{attribute 'reflection'} 
FUNCTION_BLOCK FB_Component EXTENDS FB_Cycle IMPLEMENTS I_Component
VAR_INPUT
	fbInfo:						FB_Info(sInstancePath);
	fbObserver:					FB_Observer;
	fbEvent:					FB_Event(THIS^);
END_VAR
VAR_OUTPUT
END_VAR
VAR
    {attribute 'hide'}
	{attribute 'instance-path'} 
    {attribute 'noinit'}
    sInstancePath:				STRING(255);	
	eRequest:					E_Request;
	eState:						E_State;
    {attribute 'hide'}
	eStatePrevious:				E_State;
END_VAR

METHOD PROTECTED M_Aborted : BOOL
VAR_INPUT
END_VAR
// State Aborted
M_Aborted:= True;
END_METHOD

METHOD PROTECTED M_Aborting : BOOL
VAR_INPUT
END_VAR
// State Aborting
M_Aborting:= True;
END_METHOD

METHOD PROTECTED M_Completed : BOOL
VAR_INPUT
END_VAR
// State Complete
M_Completed:= TRUE;
END_METHOD

METHOD PROTECTED M_Completing : BOOL
VAR_INPUT
END_VAR
// State Completing
M_Completing:= True;
END_METHOD

METHOD PUBLIC M_Cycle
VAR_INPUT
END_VAR
fbInfo();
fbObserver();
fbEvent();

// Handle Module Type Package states
CASE eState OF
	E_State.Undefined:
		IF M_Initialise() THEN
			eState:= E_State.Idle;					
		END_IF
		
	E_State.Resetting:
		CASE eRequest OF
			E_Request.Stop:
				eState:= E_State.Stopping;					
			E_Request.Abort:
				eState:= E_State.Aborting;						
		END_CASE	
		IF M_Resetting() THEN
			eState:= E_State.Idle;
		END_IF
		
	E_State.Idle:
		CASE eRequest OF
			E_Request.Start:
				eState:= E_State.Starting;
			E_Request.Stop:
				eState:= E_State.Stopping;					
			E_Request.Abort:
				eState:= E_State.Aborting;
			ELSE
				eRequest:= E_Request.Undefined;						
		END_CASE
		M_Idle();
		
	E_State.Starting:
		CASE eRequest OF
			E_Request.Stop:
				eState:= E_State.Stopping;					
			E_Request.Abort:
				eState:= E_State.Aborting;				
		END_CASE	
		IF M_Starting() THEN
			eState:= E_State.Execute;	
		END_IF		

	E_State.Execute:
		CASE eRequest OF
			E_Request.Pause:
				eState:= E_State.Pausing;		
			E_Request.Hold:
				eState:= E_State.Holding;		
			E_Request.Stop:
				eState:= E_State.Stopping;					
			E_Request.Abort:
				eState:= E_State.Aborting;
			ELSE
				eRequest:= E_Request.Undefined;						
		END_CASE
		IF M_Execute() THEN
			CASE eRequest OF
				E_Request.Complete:
					eState:= E_State.Completing;
			END_CASE	
		END_IF
		
	E_State.Stopping:
		CASE eRequest OF	
			E_Request.Abort:
				eState:= E_State.Aborting;			
		END_CASE	
		IF M_Stopping() THEN
			eState:= E_State.Stopped;
		END_IF

	E_State.Stopped:
		IF M_Stopped() THEN
			CASE eRequest OF
				E_Request.Reset:
					eState:= E_State.Resetting;
				ELSE
					eRequest:= E_Request.Undefined;	
			END_CASE		
		END_IF
		
	E_State.Aborting:
		IF M_Aborting() THEN
			eState:= E_State.Aborted;
		END_IF
		
	E_State.Aborted:
		IF M_Aborted() THEN
			CASE eRequest OF
				E_Request.Reset:
					eState:= E_State.Resetting;
				ELSE
					eRequest:= E_Request.Undefined;		
			END_CASE
		END_IF
		
	E_State.Pausing:
		CASE eRequest OF
			E_Request.Stop:
				eState:= E_State.Stopping;					
			E_Request.Abort:
				eState:= E_State.Aborting;					
		END_CASE	
		IF M_Pausing() THEN
			eState:= E_State.Paused;
		END_IF
	
	E_State.Paused:
		CASE eRequest OF
			E_Request.Stop:
				eState:= E_State.Stopping;					
			E_Request.Abort:
				eState:= E_State.Aborting;
			ELSE
				eRequest:= E_Request.Undefined;					
		END_CASE	
		IF M_Paused() THEN
			eState:= E_State.Resuming;			
		END_IF	
		
	E_State.Resuming:
		CASE eRequest OF
			E_Request.Stop:
				eState:= E_State.Stopping;					
			E_Request.Abort:
				eState:= E_State.Aborting;					
		END_CASE
		IF M_Resuming() THEN
			eState:= E_State.Execute;
		END_IF

	E_State.Holding:
		CASE eRequest OF
			E_Request.Stop:
				eState:= E_State.Stopping;					
			E_Request.Abort:
				eState:= E_State.Aborting;						
		END_CASE
		IF M_Holding() THEN
			eState:= E_State.Held;
		END_IF

	E_State.Held:
		CASE eRequest OF
			E_Request.Stop:
				eState:= E_State.Stopping;					
			E_Request.Abort:
				eState:= E_State.Aborting;
			ELSE
				eRequest:= E_Request.Undefined;					
		END_CASE
		IF M_Held() THEN
			eState:= E_State.Unholding;			
		END_IF	
		
	E_State.Unholding:
		CASE eRequest OF
			E_Request.Stop:
				eState:= E_State.Stopping;					
			E_Request.Abort:
				eState:= E_State.Aborting;							
		END_CASE
		IF M_Unholding() THEN
			eState:= E_State.Execute;
		END_IF
		
	E_State.Completing:
		CASE eRequest OF
			E_Request.Stop:
				eState:= E_State.Stopping;					
			E_Request.Abort:
				eState:= E_State.Aborting;				
		END_CASE
		IF M_Completing() THEN
			eState:= E_State.Completed;
		END_IF
		
	E_State.Completed:
		CASE eRequest OF
			E_Request.Stop:
				eState:= E_State.Stopping;					
			E_Request.Abort:
				eState:= E_State.Aborting;
			ELSE
				eRequest:= E_Request.Undefined;				
		END_CASE
		IF M_Completed() THEN
			CASE eRequest OF
				E_Request.Reset:	
					eState:= E_State.Resetting;
			END_CASE
		END_IF
		
	
END_CASE

CASE eState OF
	E_State.Aborted, E_State.Stopped, E_State.Completed:;
ELSE		
	this^.M_Running();
END_CASE

// Detect state changed
IF eStatePrevious <> eState THEN
	fbObserver.M_Notify(eState);
	eStatePrevious:= eState;
	M_OnStateChanged();
END_IF
END_METHOD

METHOD PROTECTED M_Execute : BOOL
VAR_INPUT
END_VAR
// State Execute
M_Execute:= TRUE;
END_METHOD

METHOD PROTECTED M_Held : BOOL
VAR_INPUT
END_VAR
// State Held
M_Held:= TRUE;
END_METHOD

METHOD PROTECTED M_Holding : BOOL
VAR_INPUT
END_VAR
// State Holding
M_Holding:= True;
END_METHOD

METHOD PROTECTED M_Idle : BOOL
VAR_INPUT
END_VAR
// State Idle
END_METHOD

METHOD PROTECTED M_Initialise : BOOL;
VAR_INPUT
END_VAR
// State Undefined
M_Initialise:= True;
END_METHOD

METHOD PUBLIC M_OnNotify
VAR_INPUT
	eState:				E_State;
END_VAR
CASE eState OF
	E_State.Undefined:;
	E_State.Idle:;
	E_State.Starting:
		M_Request(E_Request.Start);
	E_State.Execute:;
	E_State.Pausing:
		M_Request(E_Request.Pause);
	E_State.Paused:;
	E_State.Resuming:;
	E_State.Holding:
		M_Request(E_Request.Hold);
	E_State.Held:;
	E_State.Unholding:;
	E_State.Completing:
		M_Request(E_Request.Complete);
	E_State.Completed:;
	E_State.Stopping:
		M_Request(E_Request.Stop);
	E_State.Stopped:;
	E_State.Aborting:
		M_Request(E_Request.Abort);
	E_State.Aborted:;
	E_State.Resetting:
		M_Request(E_Request.Reset);
END_CASE
END_METHOD

METHOD PROTECTED M_OnStateChanged : BOOL
VAR_INPUT
END_VAR
END_METHOD

METHOD PROTECTED M_Paused : BOOL
VAR_INPUT
END_VAR
// State Held
M_Paused:= TRUE;
END_METHOD

METHOD PROTECTED M_Pausing : BOOL
VAR_INPUT
END_VAR
// State Holding
M_Pausing:= True;
END_METHOD

METHOD PUBLIC M_Request : BOOL
VAR_INPUT
	eRequest:	E_Request;
END_VAR
THIS^.eRequest:= eRequest;
CASE eRequest OF
	E_Request.Undefined:
		M_Request:= TRUE;
    E_Request.Start:
		M_Request:= eState = E_State.Execute;
    E_Request.Pause:
		IF 	fbEvent.bIngorePause THEN
			M_Request:= TRUE;
		ELSE
			M_Request:= eState = E_State.Paused;
		END_IF
    E_Request.Hold:
		IF 	fbEvent.bIngoreHold THEN
			M_Request:= TRUE;
		ELSE
			M_Request:= eState = E_State.Held;		
		END_IF
		
	E_Request.Complete:
		M_Request:= eState = E_State.Completed;	
    E_Request.Stop:
		M_Request:= eState = E_State.Stopped;	
	E_Request.Abort:
		M_Request:= eState = E_State.Aborted;	
	E_Request.Reset:
		M_Request:= eState = E_State.Idle;		

END_CASE
END_METHOD

METHOD PROTECTED M_Resetting : BOOL
VAR_INPUT
END_VAR
// State Resetting
M_Resetting:= True;
END_METHOD

METHOD PROTECTED M_Resuming : BOOL
VAR_INPUT
END_VAR
// State Holding
M_Resuming:= True;
END_METHOD

METHOD PROTECTED M_Running
VAR_INPUT
END_VAR
END_METHOD

METHOD PROTECTED M_Starting : BOOL
VAR_INPUT
END_VAR
// State Starting
M_Starting:= True;
END_METHOD

METHOD PROTECTED M_Stopped : BOOL
VAR_INPUT
END_VAR
// State Stopped
M_Stopped:= True;
END_METHOD

METHOD PROTECTED M_Stopping : BOOL
VAR_INPUT
END_VAR
// State Stopping
M_Stopping:= True;
END_METHOD

METHOD PROTECTED M_Unholding : BOOL
VAR_INPUT
END_VAR
// State Holding
M_Unholding:= True;
END_METHOD

PROPERTY PUBLIC P_Event : I_Event
GET
P_Event:= fbEvent;
END_GET
END_PROPERTY

PROPERTY PUBLIC P_Info : I_Info
GET
P_Info:= fbInfo;
END_GET
END_PROPERTY

PROPERTY PUBLIC P_Observer : I_Observer
GET
P_Observer:= fbObserver;
END_GET
END_PROPERTY

PROPERTY PUBLIC P_State : E_State
GET
P_State:= eState;
END_GET
END_PROPERTY

END_FUNCTION_BLOCK

(* stored: Version 1.1.0.1
   POU FB_Component: Id {4a8fdfc8-695a-4bb4-a889-b0289c0a194c}, SpecialFunc None
   Folder States: Id {bb7123de-6478-4234-9ee4-651df2b9bc25}
   Folder Abort: Id {4cfd24e7-9cc4-4ac8-b9a2-2bb8efd40b81}
   Folder Complete: Id {8cc75b46-b5cb-4c11-be2d-3277ffea828d}
   Folder Hold: Id {9a0b22b2-44e2-4e39-8bcb-b51e4e344ca7}
   Folder Pause: Id {9c64081e-f728-491d-9769-ffa7f6354111}
   Folder Reset: Id {fd96e000-8a80-4649-938a-5a51a16ea269}
   Folder Start: Id {3013ace2-54b5-4b17-b0c9-5400c34587df}
   Folder Stop: Id {a8159361-68bf-4749-870a-300243097586}
   Method M_Aborted: Id {851e7e88-c79a-42ec-971c-1651bbdcd922}
   Method M_Aborting: Id {2544540d-284d-4bb6-9092-9fb2d57b609d}
   Method M_Completed: Id {36dec38b-240d-4516-a167-d73475e82b56}
   Method M_Completing: Id {d7947499-dc81-4824-8eb2-1f31346a18c9}
   Method M_Cycle: Id {f033fb8d-b449-41cf-8e0e-ae093b3ee161}
   Method M_Execute: Id {7b4271f8-8ab7-4ecd-8059-762441f55350}
   Method M_Held: Id {897a0d48-e739-4f14-8313-6cf76e869ecc}
   Method M_Holding: Id {7537786e-be59-43f8-af14-91fbd68626c4}
   Method M_Idle: Id {9f0f7190-6eb5-4f18-a951-5893e9af72d3}
   Method M_Initialise: Id {54f2b561-b89f-47f6-a504-ad1a94f7dafa}
   Method M_OnNotify: Id {a99268d9-5398-44f2-992c-940f05706df3}
   Method M_OnStateChanged: Id {fed7d462-efbd-4bae-956c-60dd99530457}
   Method M_Paused: Id {5d4d1306-287a-427e-996c-3f6f19decdf3}
   Method M_Pausing: Id {b5cecc19-abeb-4b4a-b774-79fca9276a1d}
   Method M_Request: Id {ccb3d941-e869-469e-bebe-469135ac244b}
   Method M_Resetting: Id {ef3b38ac-7092-48f4-bd93-3280fba28638}
   Method M_Resuming: Id {f07a95d3-345e-4dd9-ba39-0e5ed2af03d7}
   Method M_Running: Id {b0e728db-ca35-4629-abea-b5b6a70abf0b}
   Method M_Starting: Id {0a285b28-e7e5-4050-bddf-636ff865dc31}
   Method M_Stopped: Id {3035f166-5ee3-4891-8715-c804b18a321e}
   Method M_Stopping: Id {044bf6dd-28e6-4ae0-8f4c-d70b321a375a}
   Method M_Unholding: Id {498cf474-9c66-43f0-b599-499b1410052f}
   Property P_Event: Id {3b935d9d-6278-4dc9-a359-4ee7f1c69123}
   Get Get: Id {29792270-b47c-4141-a645-41c0781f774b}
   Property P_Info: Id {6e421f29-8ecf-4944-bc3a-6ca6205a23ab}
   Get Get: Id {f1bd3bb2-b46e-4fac-8458-ce900be7323b}
   Property P_Observer: Id {2b4a3b9d-02d6-46ef-a830-8f731a2ada59}
   Get Get: Id {d2313d10-2a66-4a0c-9a20-b577c055dab4}
   Property P_State: Id {c747533f-000a-4f36-b4ba-f00b2fbb73f7}
   Get Get: Id {88d67c77-472d-4a63-bef7-c9cec62b2136} *)
